// TIA Portal V17 export
// export: Created 2023-12-22T15:04:41.9860431Z, ExportSetting WithDefaults, DisplayName Totally Integrated Automation Portal, DisplayVersion V17, DisplayName TIA Portal Openness, DisplayVersion V17, DisplayName TIA Portal Version Control Interface, DisplayVersion V17, DisplayName STEP 7 Professional, DisplayVersion V17, DisplayName STEP 7 Safety, DisplayVersion V17, DisplayName WinCC Advanced, DisplayVersion V17
DATA_BLOCK "AIx_DB"   // DB220
VERSION : 0.1
// stored: AutoNumber false, DBAccessibleFromOPCUA true, InstanceOfName AIx, InstanceOfType FB
"AIx"
   // VAR RETAIN
   //    Time_DTL { S7_SetPoint := 'True'} : DTL := DTL#2012-01-22-23:24:11.170566;
   // END_VAR
BEGIN
END_DATA_BLOCK
